{attribute addProperty BoxType "EL6201-0000-0017"}
{attribute addProperty Id "Slave_31A_DI0BIT10.125241Slave_31A_DI1BIT10.125242Slave_31A_DI2BIT10.125243Slave_31A_DI3BIT10.125244Slave_31B_DI0BIT10.125245Slave_31B_DI1BIT10.125246Slave_31B_DI2BIT10.125247Slave_31B_DI3BIT10.125248"}
{attribute addProperty CRC "3594953129"}
{attribute addProperty SizeInBites "8"}
{attribute addProperty SizeInBytes "1"}
TYPE Slave_31_Inputs_D646A1A9 :
STRUCT
	{attribute addProperty Name "Slave_31A_DI0"}
	Slave_31A_DI0 : BIT;
	{attribute addProperty Name "Slave_31A_DI1"}
	Slave_31A_DI1 : BIT;
	{attribute addProperty Name "Slave_31A_DI2"}
	Slave_31A_DI2 : BIT;
	{attribute addProperty Name "Slave_31A_DI3"}
	Slave_31A_DI3 : BIT;
	{attribute addProperty Name "Slave_31B_DI0"}
	Slave_31B_DI0 : BIT;
	{attribute addProperty Name "Slave_31B_DI1"}
	Slave_31B_DI1 : BIT;
	{attribute addProperty Name "Slave_31B_DI2"}
	Slave_31B_DI2 : BIT;
	{attribute addProperty Name "Slave_31B_DI3"}
	Slave_31B_DI3 : BIT;
END_STRUCT
END_TYPE

(* stored: Version 1.2.0.0, ProductVersion 3.1.4024.9
   DUT Slave_31_Inputs_D646A1A9: Id {9504f20a-2ea6-440a-8d8b-43d10792a747} *)
